RoboDK station: Sheet B.rdk

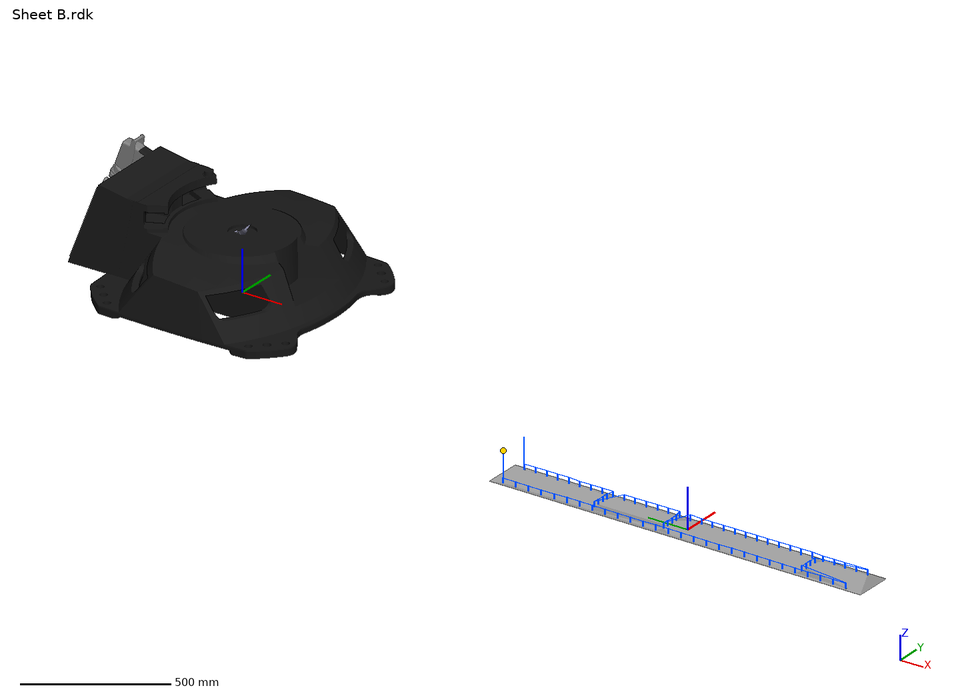
[picture v0: the station drawn from its stored meshes, robots at their saved joint values, targets as dots, program paths as lines]
Station Sheet B (saved by RoboDK 5.2.3). Poses are relative to the parent item; angles as X-Y-Z fixed-axis rotations.
  - frame KUKA KR 210 R2700 extra Base at (0, 0, 0) mm
    - robot KUKA KR 210 R2700 extra: 6 axes, payload 210 kg, reach 2696 mm, repeatability 0.06 mm, weight 1068 kg
        joint limits [-185, -140, -120, -350, -125, -350] to [185, -5, 155, 350, 125, 350]; home [0, -90, 90, 0, 0, 0]; saved at [-4.299, -27.561, 142.534, -183.011, 63.926, -182.019]
      - tool Spindle, TCP at (32, 0, 260) mm, rotated rx 0 ry 39 rz 0 deg, size 157.3 x 72 x 259.9 mm
  - frame Frame 2 at (1800, 0, -372.68) mm, rotated rx 0 ry 0 rz 90 deg
    - object Box 1 - Sheet B at (0, 0, 0) mm, size 148.8 x 1500 x 0.8 mm, geometry from Box 1 - Sheet B.stl
    - object Sheet B-box 1 Hole positioning at (0, 0, 0) mm, 72 curves, geometry from Point 72
  - machining project Point settings: rotZ(0) | rotX(0)*rotY(0) | rotz(0) | onStart | onPathStart | onApproach | onPoint | onRetract | onFinish | SetRPM(%1) | SetTool(%1) | Extruder(%1) | default | default | OutOnMov(%1) | OutOffMov(%1) | onPathFinish | M_RunCode(%1)
  - program Point (371 instructions, listed below)
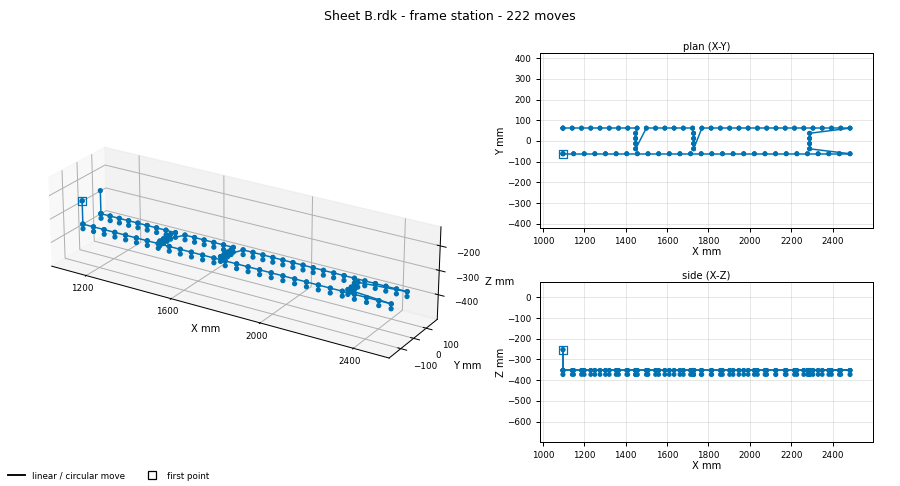
[picture p0: tool path of Sheet B.rdk in frame station, 222 of 222 moves have a stored position in this frame; points joined in program order, loops and branches not executed]

--- program Point (robot KUKA KR 210 R2700 extra) ---
  Smooth(1)
  Set speed (1000.0 mm/s)
  Set Ref.: Frame 2
  Set Tool: Spindle
  Show Spindle
  MoveJ 1 to (-61.9, 702.57, 120) mm, rotated rx 180 ry 0 rz 90 deg; joints [4.299, -27.561, 142.534, -176.989, 63.926, -177.981]
  MoveL 2 to (-61.9, 702.57, 120) mm, rotated rx 180 ry 0 rz 90 deg; joints [4.299, -27.561, 142.534, -176.989, 63.926, -177.981]
  MoveL 3 to (-61.9, 702.57, 20) mm, rotated rx -180 ry 0 rz 90 deg; joints [4.299, -20.368, 138.524, -177.064, 67.105, -177.799]
  MoveL 4 to (-61.9, 702.57, 20) mm, rotated rx -180 ry 0 rz 90 deg; joints [4.299, -20.368, 138.524, -177.064, 67.105, -177.799]
  Set speed (50.0 mm/s)
  MoveL 5 to (-61.9, 702.57, 0) mm, rotated rx 180 ry 0 rz 90 deg; joints [4.299, -19.028, 137.686, -177.075, 67.605, -177.771]
  MoveL 6 to (-61.9, 702.57, 20) mm, rotated rx -180 ry 0 rz 90 deg; joints [4.299, -20.368, 138.524, -177.064, 67.105, -177.799]
  Set speed (1000.0 mm/s)
  MoveL 7 to (-61.9, 651.24, 20) mm, rotated rx 180 ry 0 rz 90 deg; joints [4.048, -22.239, 136.879, -177.157, 63.598, -178.117]
  Set speed (50.0 mm/s)
  MoveL 8 to (-61.9, 651.24, 0) mm, rotated rx -180 ry 0 rz 90 deg; joints [4.048, -20.899, 136.068, -177.17, 64.126, -178.088]
  MoveL 9 to (-61.9, 651.24, 20) mm, rotated rx 180 ry 0 rz 90 deg; joints [4.048, -22.239, 136.879, -177.157, 63.598, -178.117]
  Set speed (1000.0 mm/s)
  MoveL 10 to (-61.9, 599.91, 20) mm, rotated rx 180 ry 0 rz 90 deg; joints [3.824, -23.844, 135.126, -177.229, 60.248, -178.402]
  Set speed (50.0 mm/s)
  MoveL 11 to (-61.9, 599.91, 0) mm, rotated rx -180 ry 0 rz 90 deg; joints [3.824, -22.512, 134.341, -177.244, 60.795, -178.372]
  MoveL 12 to (-61.9, 599.91, 20) mm, rotated rx 180 ry 0 rz 90 deg; joints [3.824, -23.844, 135.126, -177.229, 60.248, -178.402]
  Set speed (1000.0 mm/s)
  MoveL 13 to (-61.9, 548.57, 20) mm, rotated rx -180 ry 0 rz 90 deg; joints [3.624, -25.203, 133.273, -177.283, 57.044, -178.661]
  Set speed (50.0 mm/s)
  MoveL 14 to (-61.9, 548.57, 0) mm, rotated rx 180 ry 0 rz 90 deg; joints [3.624, -23.885, 132.514, -177.3, 57.602, -178.63]
  MoveL 15 to (-61.9, 548.57, 20) mm, rotated rx -180 ry 0 rz 90 deg; joints [3.624, -25.203, 133.273, -177.283, 57.044, -178.661]
  Set speed (1000.0 mm/s)
  MoveL 16 to (-61.9, 497.24, 20) mm, rotated rx 180 ry 0 rz 90 deg; joints [3.444, -26.333, 131.329, -177.321, 53.975, -178.899]
  Set speed (50.0 mm/s)
  MoveL 17 to (-61.9, 497.24, 0) mm, rotated rx -180 ry 0 rz 90 deg; joints [3.444, -25.033, 130.594, -177.34, 54.539, -178.866]
  MoveL 18 to (-61.9, 497.24, 20) mm, rotated rx 180 ry 0 rz 90 deg; joints [3.444, -26.333, 131.329, -177.321, 53.975, -178.899]
  Set speed (1000.0 mm/s)
  MoveL 19 to (-61.9, 445.91, 20) mm, rotated rx 180 ry 0 rz 90 deg; joints [3.28, -27.254, 129.3, -177.345, 51.03, -179.12]
  Set speed (50.0 mm/s)
  MoveL 20 to (-61.9, 445.91, 0) mm, rotated rx 180 ry 0 rz 90 deg; joints [3.28, -25.976, 128.588, -177.366, 51.595, -179.087]
  MoveL 21 to (-61.9, 445.91, 20) mm, rotated rx 180 ry 0 rz 90 deg; joints [3.28, -27.254, 129.3, -177.345, 51.03, -179.12]
  Set speed (1000.0 mm/s)
  MoveL 22 to (-61.9, 394.57, 20) mm, rotated rx -180 ry 0 rz 90 deg; joints [3.132, -27.982, 127.19, -177.357, 48.196, -179.328]
  Set speed (50.0 mm/s)
  MoveL 23 to (-61.9, 394.57, 0) mm, rotated rx 180 ry 0 rz 90 deg; joints [3.132, -26.729, 126.5, -177.379, 48.759, -179.294]
  MoveL 24 to (-61.9, 394.57, 20) mm, rotated rx -180 ry 0 rz 90 deg; joints [3.132, -27.982, 127.19, -177.357, 48.196, -179.328]
  Set speed (1000.0 mm/s)
  MoveL 25 to (-61.9, 343.24, 20) mm, rotated rx -180 ry 0 rz 90 deg; joints [2.996, -28.534, 125.006, -177.355, 45.464, -179.526]
  Set speed (50.0 mm/s)
  MoveL 26 to (-61.9, 343.24, 0) mm, rotated rx 180 ry 0 rz 90 deg; joints [2.996, -27.307, 124.335, -177.38, 46.02, -179.491]
  MoveL 27 to (-61.9, 343.24, 20) mm, rotated rx -180 ry 0 rz 90 deg; joints [2.996, -28.534, 125.006, -177.355, 45.464, -179.526]
  Set speed (1000.0 mm/s)
  MoveL 28 to (-61.9, 291.91, 20) mm, rotated rx -180 ry 0 rz 90 deg; joints [2.872, -28.924, 122.749, -177.341, 42.821, -179.718]
  Set speed (50.0 mm/s)
  MoveL 29 to (-61.9, 291.91, 0) mm, rotated rx 180 ry 0 rz 90 deg; joints [2.872, -27.723, 122.097, -177.369, 43.369, -179.681]
  MoveL 30 to (-61.9, 291.91, 20) mm, rotated rx -180 ry 0 rz 90 deg; joints [2.872, -28.924, 122.749, -177.341, 42.821, -179.718]
  Set speed (1000.0 mm/s)
  MoveL 31 to (-61.9, 240.57, 20) mm, rotated rx -180 ry 0 rz 90 deg; joints [2.757, -29.164, 120.423, -177.315, 40.257, -179.906]
  Set speed (50.0 mm/s)
  MoveL 32 to (-61.9, 240.57, 0) mm, rotated rx -180 ry 0 rz 90 deg; joints [2.757, -27.991, 119.788, -177.344, 40.795, -179.868]
  MoveL 33 to (-61.9, 240.57, 20) mm, rotated rx -180 ry 0 rz 90 deg; joints [2.757, -29.164, 120.423, -177.315, 40.257, -179.906]
  Set speed (1000.0 mm/s)
  MoveL 34 to (-61.9, 189.24, 20) mm, rotated rx 180 ry 0 rz 90 deg; joints [2.651, -29.267, 118.029, -177.275, 37.764, -180.093]
  Set speed (50.0 mm/s)
  MoveL 35 to (-61.9, 189.24, 0) mm, rotated rx -180 ry 0 rz 90 deg; joints [2.651, -28.12, 117.41, -177.307, 38.291, -180.053]
  MoveL 36 to (-61.9, 189.24, 20) mm, rotated rx 180 ry 0 rz 90 deg; joints [2.651, -29.267, 118.029, -177.275, 37.764, -180.093]
  Set speed (1000.0 mm/s)
  MoveL 37 to (-61.9, 137.91, 20) mm, rotated rx -180 ry 0 rz 90 deg; joints [2.553, -29.241, 115.568, -177.221, 35.331, -180.283]
  Set speed (50.0 mm/s)
  MoveL 38 to (-61.9, 137.91, 0) mm, rotated rx -180 ry 0 rz 90 deg; joints [2.553, -28.121, 114.963, -177.256, 35.846, -180.24]
  MoveL 39 to (-61.9, 137.91, 20) mm, rotated rx -180 ry 0 rz 90 deg; joints [2.553, -29.241, 115.568, -177.221, 35.331, -180.283]
  Set speed (1000.0 mm/s)
  MoveL 40 to (-61.9, 86.57, 20) mm, rotated rx 180 ry 0 rz 90 deg; joints [2.462, -29.097, 113.041, -177.151, 32.95, -180.478]
  Set speed (50.0 mm/s)
  MoveL 41 to (-61.9, 86.57, 0) mm, rotated rx -180 ry 0 rz 90 deg; joints [2.462, -28.002, 112.448, -177.188, 33.452, -180.432]
  MoveL 42 to (-61.9, 86.57, 20) mm, rotated rx 180 ry 0 rz 90 deg; joints [2.462, -29.097, 113.041, -177.151, 32.95, -180.478]
  Set speed (1000.0 mm/s)
  MoveL 43 to (-61.9, 35.24, 20) mm, rotated rx 180 ry 0 rz 90 deg; joints [2.378, -28.841, 110.446, -177.061, 30.614, -180.681]
  Set speed (50.0 mm/s)
  MoveL 44 to (-61.9, 35.24, 0) mm, rotated rx -180 ry 0 rz 90 deg; joints [2.378, -27.771, 109.865, -177.103, 31.102, -180.633]
  MoveL 45 to (-61.9, 35.24, 20) mm, rotated rx 180 ry 0 rz 90 deg; joints [2.378, -28.841, 110.446, -177.061, 30.614, -180.681]
  Set speed (1000.0 mm/s)
  MoveL 46 to (-61.9, -16.09, 20) mm, rotated rx 180 ry 0 rz 90 deg; joints [2.299, -28.479, 107.783, -176.949, 28.315, -180.899]
  Set speed (50.0 mm/s)
  MoveL 47 to (-61.9, -16.09, 0) mm, rotated rx -180 ry 0 rz 90 deg; joints [2.299, -27.434, 107.212, -176.996, 28.789, -180.847]
  MoveL 48 to (-61.9, -16.09, 20) mm, rotated rx 180 ry 0 rz 90 deg; joints [2.299, -28.479, 107.783, -176.949, 28.315, -180.899]
  Set speed (1000.0 mm/s)
  MoveL 49 to (-61.9, -67.43, 20) mm, rotated rx 180 ry 0 rz 90 deg; joints [2.225, -28.017, 105.049, -176.811, 26.045, -181.137]
  Set speed (50.0 mm/s)
  MoveL 50 to (-61.9, -67.43, 0) mm, rotated rx -180 ry 0 rz 90 deg; joints [2.225, -26.995, 104.487, -176.862, 26.505, -181.079]
  MoveL 51 to (-61.9, -67.43, 20) mm, rotated rx 180 ry 0 rz 90 deg; joints [2.225, -28.017, 105.049, -176.811, 26.045, -181.137]
  Set speed (1000.0 mm/s)
  MoveL 52 to (-61.9, -118.76, 20) mm, rotated rx -180 ry 0 rz 90 deg; joints [2.155, -27.459, 102.241, -176.637, 23.799, -181.402]
  Set speed (50.0 mm/s)
  MoveL 53 to (-61.9, -118.76, 0) mm, rotated rx -180 ry 0 rz 90 deg; joints [2.155, -26.459, 101.687, -176.696, 24.244, -181.338]
  MoveL 54 to (-61.9, -118.76, 20) mm, rotated rx -180 ry 0 rz 90 deg; joints [2.155, -27.459, 102.241, -176.637, 23.799, -181.402]
  Set speed (1000.0 mm/s)
  MoveL 55 to (-61.9, -170.09, 20) mm, rotated rx -180 ry 0 rz 90 deg; joints [2.09, -26.809, 99.357, -176.42, 21.568, -181.705]
  Set speed (50.0 mm/s)
  MoveL 56 to (-61.9, -170.09, 0) mm, rotated rx -180 ry 0 rz 90 deg; joints [2.09, -25.829, 98.809, -176.487, 21.998, -181.633]
  MoveL 57 to (-61.9, -170.09, 20) mm, rotated rx -180 ry 0 rz 90 deg; joints [2.09, -26.809, 99.357, -176.42, 21.568, -181.705]
  Set speed (1000.0 mm/s)
  MoveL 58 to (-61.9, -221.43, 20) mm, rotated rx 180 ry 0 rz 90 deg; joints [2.029, -26.067, 96.391, -176.144, 19.346, -182.062]
  Set speed (50.0 mm/s)
  MoveL 59 to (-61.9, -221.43, 0) mm, rotated rx 180 ry 0 rz 90 deg; joints [2.029, -25.107, 95.847, -176.222, 19.762, -181.979]
  MoveL 60 to (-61.9, -221.43, 20) mm, rotated rx 180 ry 0 rz 90 deg; joints [2.029, -26.067, 96.391, -176.144, 19.346, -182.062]
  Set speed (1000.0 mm/s)
  MoveL 61 to (-61.9, -272.76, 20) mm, rotated rx -180 ry 0 rz 90 deg; joints [1.971, -25.236, 93.337, -175.785, 17.128, -182.496]
  Set speed (50.0 mm/s)
  MoveL 62 to (-61.9, -272.76, 0) mm, rotated rx -180 ry 0 rz 90 deg; joints [1.971, -24.295, 92.797, -175.879, 17.528, -182.398]
  MoveL 63 to (-61.9, -272.76, 20) mm, rotated rx -180 ry 0 rz 90 deg; joints [1.971, -25.236, 93.337, -175.785, 17.128, -182.496]
  Set speed (1000.0 mm/s)
  MoveL 64 to (-61.9, -324.09, 20) mm, rotated rx -180 ry 0 rz 90 deg; joints [1.916, -24.316, 90.189, -175.307, 14.906, -183.046]
  Set speed (50.0 mm/s)
  MoveL 65 to (-61.9, -324.09, 0) mm, rotated rx -180 ry 0 rz 90 deg; joints [1.916, -23.391, 89.651, -175.423, 15.29, -182.926]
  MoveL 66 to (-61.9, -324.09, 20) mm, rotated rx -180 ry 0 rz 90 deg; joints [1.916, -24.316, 90.189, -175.307, 14.906, -183.046]
  Set speed (1000.0 mm/s)
  MoveL 67 to (-61.9, -375.43, 20) mm, rotated rx 180 ry 0 rz 90 deg; joints [1.865, -23.305, 86.938, -174.644, 12.672, -183.777]
  Set speed (50.0 mm/s)
  MoveL 68 to (-61.9, -375.43, 0) mm, rotated rx -180 ry 0 rz 90 deg; joints [1.865, -22.396, 86.4, -174.793, 13.041, -183.624]
  MoveL 69 to (-61.9, -375.43, 20) mm, rotated rx 180 ry 0 rz 90 deg; joints [1.865, -23.305, 86.938, -174.644, 12.672, -183.777]
  Set speed (1000.0 mm/s)
  MoveL 70 to (-61.9, -426.76, 20) mm, rotated rx -180 ry 0 rz 90 deg; joints [1.816, -22.202, 83.574, -173.671, 10.421, -184.814]
  Set speed (50.0 mm/s)
  MoveL 71 to (-61.9, -426.76, 0) mm, rotated rx 180 ry 0 rz 90 deg; joints [1.816, -21.307, 83.035, -173.877, 10.774, -184.605]
  MoveL 72 to (-61.9, -426.76, 20) mm, rotated rx -180 ry 0 rz 90 deg; joints [1.816, -22.202, 83.574, -173.671, 10.421, -184.814]
  Set speed (1000.0 mm/s)
  MoveL 73 to (-61.9, -478.09, 20) mm, rotated rx 180 ry 0 rz 90 deg; joints [1.769, -21.002, 80.085, -172.118, 8.145, -186.428]
  Set speed (50.0 mm/s)
  MoveL 74 to (-61.9, -478.09, 0) mm, rotated rx -180 ry 0 rz 90 deg; joints [1.769, -20.12, 79.541, -172.43, 8.481, -186.113]
  MoveL 75 to (-61.9, -478.09, 20) mm, rotated rx 180 ry 0 rz 90 deg; joints [1.769, -21.002, 80.085, -172.118, 8.145, -186.428]
  Set speed (1000.0 mm/s)
  MoveL 76 to (-61.9, -529.43, 20) mm, rotated rx -180 ry 0 rz 90 deg; joints [1.725, -19.7, 76.453, -169.273, 5.842, -189.332]
  Set speed (50.0 mm/s)
  MoveL 77 to (-61.9, -529.43, 0) mm, rotated rx 180 ry 0 rz 90 deg; joints [1.725, -18.828, 75.903, -169.828, 6.158, -188.774]
  MoveL 78 to (-61.9, -529.43, 20) mm, rotated rx -180 ry 0 rz 90 deg; joints [1.725, -19.7, 76.453, -169.273, 5.842, -189.332]
  Set speed (1000.0 mm/s)
  MoveL 79 to (-61.9, -580.76, 20) mm, rotated rx -180 ry 0 rz 90 deg; joints [1.683, -18.288, 72.66, -162.494, 3.523, -196.167]
  Set speed (50.0 mm/s)
  MoveL 80 to (-61.9, -580.76, 0) mm, rotated rx 180 ry 0 rz 90 deg; joints [1.683, -17.425, 72.101, -163.866, 3.814, -194.792]
  MoveL 81 to (-61.9, -580.76, 20) mm, rotated rx -180 ry 0 rz 90 deg; joints [1.683, -18.288, 72.66, -162.494, 3.523, -196.167]
  Set speed (1000.0 mm/s)
  MoveL 82 to (-61.9, -632.09, 20) mm, rotated rx -180 ry 0 rz 70 deg; joints [-0.839, -16.255, 67.408, -277.48, 13.05, -98.802]
  Set speed (50.0 mm/s)
  MoveL 83 to (-61.9, -632.09, 0) mm, rotated rx -180 ry 0 rz 70 deg; joints [-0.839, -15.4, 66.832, -276.285, 13.016, -100.029]
  MoveL 84 to (-61.9, -632.09, 20) mm, rotated rx -180 ry 0 rz 70 deg; joints [-0.839, -16.255, 67.408, -277.48, 13.05, -98.802]
  Set speed (1000.0 mm/s)
  MoveL 85 to (-61.9, -683.43, 20) mm, rotated rx -180 ry 0 rz 70 deg; joints [-0.819, -14.541, 63.132, -288.04, 13.606, -87.937]
  Set speed (50.0 mm/s)
  MoveL 86 to (-61.9, -683.43, 0) mm, rotated rx -180 ry 0 rz 70 deg; joints [-0.819, -13.689, 62.537, -287.023, 13.528, -88.983]
  MoveL 87 to (-61.9, -683.43, 20) mm, rotated rx -180 ry 0 rz 70 deg; joints [-0.819, -14.541, 63.132, -288.04, 13.606, -87.937]
  Set speed (1000.0 mm/s)
  MoveL 88 to (-38, -488.43, 20) mm, rotated rx 180 ry 0 rz 90 deg; joints [1.081, -20.763, 79.407, -174.897, 7.669, -184.218]
  Set speed (50.0 mm/s)
  MoveL 89 to (-38, -488.43, 0) mm, rotated rx 180 ry 0 rz 90 deg; joints [1.081, -19.883, 78.862, -175.109, 8.003, -184.003]
  MoveL 90 to (-38, -488.43, 20) mm, rotated rx -180 ry 0 rz 90 deg; joints [1.081, -20.763, 79.407, -174.897, 7.669, -184.218]
  Set speed (1000.0 mm/s)
  MoveL 91 to (-13, -488.43, 20) mm, rotated rx 180 ry 0 rz 90 deg; joints [0.37, -20.771, 79.429, -178.254, 7.661, -181.443]
  Set speed (50.0 mm/s)
  MoveL 92 to (-13, -488.43, 0) mm, rotated rx -180 ry 0 rz 90 deg; joints [0.37, -19.89, 78.884, -178.327, 7.997, -181.369]
  MoveL 93 to (-13, -488.43, 20) mm, rotated rx 180 ry 0 rz 90 deg; joints [0.37, -20.771, 79.429, -178.254, 7.661, -181.443]
  Set speed (1000.0 mm/s)
  MoveL 94 to (12, -488.43, 20) mm, rotated rx -180 ry 0 rz 90 deg; joints [-0.341, -20.771, 79.429, -181.611, 7.661, -178.668]
  Set speed (50.0 mm/s)
  MoveL 95 to (12, -488.43, 0) mm, rotated rx -180 ry 0 rz 90 deg; joints [-0.341, -19.891, 78.885, -181.544, 7.996, -178.736]
  MoveL 96 to (12, -488.43, 20) mm, rotated rx -180 ry 0 rz 90 deg; joints [-0.341, -20.771, 79.429, -181.611, 7.661, -178.668]
  Set speed (1000.0 mm/s)
  MoveL 97 to (37, -488.43, 20) mm, rotated rx -180 ry 0 rz 90 deg; joints [-1.052, -20.763, 79.408, -184.969, 7.668, -175.893]
  Set speed (50.0 mm/s)
  MoveL 98 to (37, -488.43, 0) mm, rotated rx -180 ry 0 rz 90 deg; joints [-1.052, -19.883, 78.863, -184.762, 8.003, -176.102]
  MoveL 99 to (37, -488.43, 20) mm, rotated rx -180 ry 0 rz 90 deg; joints [-1.052, -20.763, 79.408, -184.969, 7.668, -175.893]
  Set speed (1000.0 mm/s)
  MoveL 100 to (61.9, -683.43, 20) mm, rotated rx -180 ry 0 rz 70 deg; joints [-4, -14.358, 62.684, -288.833, 15.691, -89.578]
  Set speed (50.0 mm/s)
  MoveL 101 to (61.9, -683.43, 0) mm, rotated rx -180 ry 0 rz 70 deg; joints [-4, -13.506, 62.087, -287.969, 15.61, -90.475]
  MoveL 102 to (61.9, -683.43, 20) mm, rotated rx 180 ry 0 rz 70 deg; joints [-4, -14.358, 62.684, -288.833, 15.691, -89.578]
  Set speed (1000.0 mm/s)
  MoveL 103 to (61.9, -638.72, 20) mm, rotated rx -180 ry 0 rz 70 deg; joints [-4.081, -15.87, 66.435, -280.993, 15.164, -97.774]
  Set speed (50.0 mm/s)
  MoveL 104 to (61.9, -638.72, 0) mm, rotated rx -180 ry 0 rz 70 deg; joints [-4.081, -15.016, 65.855, -279.998, 15.114, -98.805]
  MoveL 105 to (61.9, -638.72, 20) mm, rotated rx -180 ry 0 rz 70 deg; joints [-4.081, -15.87, 66.435, -280.993, 15.164, -97.774]
  Set speed (1000.0 mm/s)
  MoveL 106 to (61.9, -594.01, 20) mm, rotated rx 180 ry 0 rz 90 deg; joints [-1.672, -17.905, 71.652, -201.052, 2.931, -160.273]
  Set speed (50.0 mm/s)
  MoveL 107 to (61.9, -594.01, 0) mm, rotated rx -180 ry 0 rz 90 deg; joints [-1.672, -17.044, 71.09, -199.137, 3.212, -162.191]
  MoveL 108 to (61.9, -594.01, 20) mm, rotated rx -180 ry 0 rz 90 deg; joints [-1.672, -17.905, 71.652, -201.052, 2.931, -160.273]
  Set speed (1000.0 mm/s)
  MoveL 109 to (61.9, -549.3, 20) mm, rotated rx 180 ry 0 rz 90 deg; joints [-1.709, -19.167, 75.005, -192.575, 4.944, -168.798]
  Set speed (50.0 mm/s)
  MoveL 110 to (61.9, -549.3, 0) mm, rotated rx 180 ry 0 rz 90 deg; joints [-1.709, -18.299, 74.452, -191.829, 5.252, -169.547]
  MoveL 111 to (61.9, -549.3, 20) mm, rotated rx 180 ry 0 rz 90 deg; joints [-1.709, -19.167, 75.005, -192.575, 4.944, -168.798]
  Set speed (1000.0 mm/s)
  MoveL 112 to (61.9, -504.59, 20) mm, rotated rx -180 ry 0 rz 90 deg; joints [-1.746, -20.343, 78.229, -189.105, 6.96, -172.318]
  Set speed (50.0 mm/s)
  MoveL 113 to (61.9, -504.59, 0) mm, rotated rx 180 ry 0 rz 90 deg; joints [-1.746, -19.466, 77.682, -188.697, 7.286, -172.729]
  MoveL 114 to (61.9, -504.59, 20) mm, rotated rx -180 ry 0 rz 90 deg; joints [-1.746, -20.343, 78.229, -189.105, 6.96, -172.318]
  Set speed (1000.0 mm/s)
  MoveL 115 to (61.9, -459.88, 20) mm, rotated rx -180 ry 0 rz 90 deg; joints [-1.785, -21.439, 81.338, -187.236, 8.956, -174.239]
  Set speed (50.0 mm/s)
  MoveL 116 to (61.9, -459.88, 0) mm, rotated rx 180 ry 0 rz 90 deg; joints [-1.785, -20.552, 80.796, -186.971, 9.298, -174.508]
  MoveL 117 to (61.9, -459.88, 20) mm, rotated rx -180 ry 0 rz 90 deg; joints [-1.785, -21.439, 81.338, -187.236, 8.956, -174.239]
  Set speed (1000.0 mm/s)
  MoveL 118 to (61.9, -415.17, 20) mm, rotated rx 180 ry 0 rz 90 deg; joints [-1.826, -22.459, 84.344, -186.072, 10.931, -175.457]
  Set speed (50.0 mm/s)
  MoveL 119 to (61.9, -415.17, 0) mm, rotated rx -180 ry 0 rz 90 deg; joints [-1.826, -21.561, 83.805, -185.882, 11.288, -175.651]
  MoveL 120 to (61.9, -415.17, 20) mm, rotated rx 180 ry 0 rz 90 deg; joints [-1.826, -22.459, 84.344, -186.072, 10.931, -175.457]
  Set speed (1000.0 mm/s)
  MoveL 121 to (61.9, -370.46, 20) mm, rotated rx 180 ry 0 rz 90 deg; joints [-1.87, -23.407, 87.258, -185.281, 12.889, -176.304]
  Set speed (50.0 mm/s)
  MoveL 122 to (61.9, -370.46, 0) mm, rotated rx -180 ry 0 rz 90 deg; joints [-1.87, -22.497, 86.72, -185.136, 13.259, -176.454]
  MoveL 123 to (61.9, -370.46, 20) mm, rotated rx 180 ry 0 rz 90 deg; joints [-1.87, -23.407, 87.258, -185.281, 12.889, -176.304]
  Set speed (1000.0 mm/s)
  MoveL 124 to (61.9, -325.75, 20) mm, rotated rx -180 ry 0 rz 90 deg; joints [-1.915, -24.285, 90.086, -184.711, 14.834, -176.934]
  Set speed (50.0 mm/s)
  MoveL 125 to (61.9, -325.75, 0) mm, rotated rx 180 ry 0 rz 90 deg; joints [-1.915, -23.361, 89.548, -184.594, 15.218, -177.054]
  MoveL 126 to (61.9, -325.75, 20) mm, rotated rx -180 ry 0 rz 90 deg; joints [-1.915, -24.285, 90.086, -184.711, 14.834, -176.934]
  Set speed (1000.0 mm/s)
  MoveL 127 to (61.9, -281.04, 20) mm, rotated rx -180 ry 0 rz 90 deg; joints [-1.962, -25.094, 92.836, -184.282, 16.77, -177.424]
  Set speed (50.0 mm/s)
  MoveL 128 to (61.9, -281.04, 0) mm, rotated rx 180 ry 0 rz 90 deg; joints [-1.962, -24.155, 92.296, -184.186, 17.168, -177.525]
  MoveL 129 to (61.9, -281.04, 20) mm, rotated rx -180 ry 0 rz 90 deg; joints [-1.962, -25.094, 92.836, -184.282, 16.77, -177.424]
  Set speed (1000.0 mm/s)
  MoveL 130 to (61.9, -236.33, 20) mm, rotated rx -180 ry 0 rz 90 deg; joints [-2.012, -25.835, 95.514, -183.95, 18.703, -177.821]
  Set speed (50.0 mm/s)
  MoveL 131 to (61.9, -236.33, 0) mm, rotated rx 180 ry 0 rz 90 deg; joints [-2.012, -24.881, 94.971, -183.868, 19.114, -177.908]
  MoveL 132 to (61.9, -236.33, 20) mm, rotated rx -180 ry 0 rz 90 deg; joints [-2.012, -25.835, 95.514, -183.95, 18.703, -177.821]
  Set speed (1000.0 mm/s)
  MoveL 133 to (61.9, -191.62, 20) mm, rotated rx -180 ry 0 rz 90 deg; joints [-2.064, -26.509, 98.123, -183.687, 20.636, -178.153]
  Set speed (50.0 mm/s)
  MoveL 134 to (61.9, -191.62, 0) mm, rotated rx -180 ry 0 rz 90 deg; joints [-2.064, -25.538, 97.577, -183.616, 21.06, -178.229]
  MoveL 135 to (61.9, -191.62, 20) mm, rotated rx -180 ry 0 rz 90 deg; joints [-2.064, -26.509, 98.123, -183.687, 20.636, -178.153]
  Set speed (1000.0 mm/s)
  MoveL 136 to (61.9, -146.91, 20) mm, rotated rx 180 ry 0 rz 90 deg; joints [-2.119, -27.114, 100.669, -183.475, 22.574, -178.437]
  Set speed (50.0 mm/s)
  MoveL 137 to (61.9, -146.91, 0) mm, rotated rx -180 ry 0 rz 90 deg; joints [-2.119, -26.125, 100.119, -183.413, 23.011, -178.505]
  MoveL 138 to (61.9, -146.91, 20) mm, rotated rx 180 ry 0 rz 90 deg; joints [-2.119, -27.114, 100.669, -183.475, 22.574, -178.437]
  Set speed (1000.0 mm/s)
  MoveL 139 to (61.9, -102.2, 20) mm, rotated rx -180 ry 0 rz 90 deg; joints [-2.177, -27.649, 103.155, -183.302, 24.521, -178.687]
  Set speed (50.0 mm/s)
  MoveL 140 to (61.9, -102.2, 0) mm, rotated rx -180 ry 0 rz 90 deg; joints [-2.177, -26.642, 102.599, -183.247, 24.971, -178.749]
  MoveL 141 to (61.9, -102.2, 20) mm, rotated rx -180 ry 0 rz 90 deg; joints [-2.177, -27.649, 103.155, -183.302, 24.521, -178.687]
  Set speed (1000.0 mm/s)
  MoveL 142 to (61.9, -57.49, 20) mm, rotated rx -180 ry 0 rz 90 deg; joints [-2.239, -28.114, 105.584, -183.16, 26.483, -178.911]
  Set speed (50.0 mm/s)
  MoveL 143 to (61.9, -57.49, 0) mm, rotated rx -180 ry 0 rz 90 deg; joints [-2.239, -27.088, 105.02, -183.11, 26.945, -178.967]
  MoveL 144 to (61.9, -57.49, 20) mm, rotated rx -180 ry 0 rz 90 deg; joints [-2.239, -28.114, 105.584, -183.16, 26.483, -178.911]
  Set speed (1000.0 mm/s)
  MoveL 145 to (61.9, -12.78, 20) mm, rotated rx -180 ry 0 rz 90 deg; joints [-2.304, -28.505, 107.957, -183.043, 28.463, -179.115]
  Set speed (50.0 mm/s)
  MoveL 146 to (61.9, -12.78, 0) mm, rotated rx 180 ry 0 rz 90 deg; joints [-2.304, -27.459, 107.385, -182.997, 28.937, -179.167]
  MoveL 147 to (61.9, -12.78, 20) mm, rotated rx -180 ry 0 rz 90 deg; joints [-2.304, -28.505, 107.957, -183.043, 28.463, -179.115]
  Set speed (1000.0 mm/s)
  MoveL 148 to (61.9, 31.93, 20) mm, rotated rx 180 ry 0 rz 90 deg; joints [-2.373, -28.82, 110.276, -182.945, 30.465, -179.305]
  Set speed (50.0 mm/s)
  MoveL 149 to (61.9, 31.93, 0) mm, rotated rx -180 ry 0 rz 90 deg; joints [-2.373, -27.753, 109.696, -182.903, 30.952, -179.354]
  MoveL 150 to (61.9, 31.93, 20) mm, rotated rx 180 ry 0 rz 90 deg; joints [-2.373, -28.82, 110.276, -182.945, 30.465, -179.305]
  Set speed (1000.0 mm/s)
  MoveL 151 to (-38, 71.57, 20) mm, rotated rx -180 ry 0 rz 90 deg; joints [1.497, -29.037, 112.331, -178.237, 32.296, -180.327]
  Set speed (50.0 mm/s)
  MoveL 152 to (-38, 71.57, 0) mm, rotated rx 180 ry 0 rz 90 deg; joints [1.497, -27.95, 111.742, -178.261, 32.795, -180.299]
  MoveL 153 to (-38, 71.57, 20) mm, rotated rx -180 ry 0 rz 90 deg; joints [1.497, -29.037, 112.331, -178.237, 32.296, -180.327]
  Set speed (1000.0 mm/s)
  MoveL 154 to (-13, 71.57, 20) mm, rotated rx 180 ry 0 rz 90 deg; joints [0.512, -29.039, 112.353, -179.397, 32.314, -180.112]
  Set speed (50.0 mm/s)
  MoveL 155 to (-13, 71.57, 0) mm, rotated rx -180 ry 0 rz 90 deg; joints [0.512, -27.951, 111.764, -179.405, 32.813, -180.102]
  MoveL 156 to (-13, 71.57, 20) mm, rotated rx 180 ry 0 rz 90 deg; joints [0.512, -29.039, 112.353, -179.397, 32.314, -180.112]
  Set speed (1000.0 mm/s)
  MoveL 157 to (12, 71.57, 20) mm, rotated rx 180 ry 0 rz 90 deg; joints [-0.473, -29.039, 112.353, -180.557, 32.315, -179.897]
  Set speed (50.0 mm/s)
  MoveL 158 to (12, 71.57, 0) mm, rotated rx 180 ry 0 rz 90 deg; joints [-0.473, -27.951, 111.764, -180.549, 32.813, -179.906]
  MoveL 159 to (12, 71.57, 20) mm, rotated rx 180 ry 0 rz 90 deg; joints [-0.473, -29.039, 112.353, -180.557, 32.315, -179.897]
  Set speed (1000.0 mm/s)
  MoveL 160 to (37, 71.57, 20) mm, rotated rx -180 ry 0 rz 90 deg; joints [-1.457, -29.037, 112.332, -181.717, 32.298, -179.682]
  Set speed (50.0 mm/s)
  MoveL 161 to (37, 71.57, 0) mm, rotated rx -180 ry 0 rz 90 deg; joints [-1.457, -27.95, 111.743, -181.693, 32.796, -179.709]
  MoveL 162 to (37, 71.57, 20) mm, rotated rx -180 ry 0 rz 90 deg; joints [-1.457, -29.037, 112.332, -181.717, 32.298, -179.682]
  Set speed (1000.0 mm/s)
  MoveL 163 to (61.9, 76.64, 20) mm, rotated rx 180 ry 0 rz 90 deg; joints [-2.446, -29.056, 112.544, -182.865, 32.495, -179.484]
  Set speed (50.0 mm/s)
  MoveL 164 to (61.9, 76.64, 0) mm, rotated rx -180 ry 0 rz 90 deg; joints [-2.446, -27.966, 111.954, -182.827, 32.994, -179.53]
  MoveL 165 to (61.9, 76.64, 20) mm, rotated rx 180 ry 0 rz 90 deg; joints [-2.446, -29.056, 112.544, -182.865, 32.495, -179.484]
  Set speed (1000.0 mm/s)
  MoveL 166 to (61.9, 121.35, 20) mm, rotated rx -180 ry 0 rz 90 deg; joints [-2.523, -29.207, 114.76, -182.8, 34.558, -179.655]
  Set speed (50.0 mm/s)
  MoveL 167 to (61.9, 121.35, 0) mm, rotated rx -180 ry 0 rz 90 deg; joints [-2.523, -28.096, 114.16, -182.764, 35.068, -179.699]
  MoveL 168 to (61.9, 121.35, 20) mm, rotated rx -180 ry 0 rz 90 deg; joints [-2.523, -29.207, 114.76, -182.8, 34.558, -179.655]
  Set speed (1000.0 mm/s)
  MoveL 169 to (61.9, 166.06, 20) mm, rotated rx 180 ry 0 rz 90 deg; joints [-2.606, -29.271, 116.926, -182.747, 36.658, -179.822]
  Set speed (50.0 mm/s)
  MoveL 170 to (61.9, 166.06, 0) mm, rotated rx -180 ry 0 rz 90 deg; joints [-2.606, -28.136, 116.313, -182.714, 37.18, -179.863]
  MoveL 171 to (61.9, 166.06, 20) mm, rotated rx 180 ry 0 rz 90 deg; joints [-2.606, -29.271, 116.926, -182.747, 36.658, -179.822]
  Set speed (1000.0 mm/s)
  MoveL 172 to (61.9, 210.77, 20) mm, rotated rx -180 ry 0 rz 90 deg; joints [-2.695, -29.24, 119.041, -182.706, 38.802, -179.985]
  Set speed (50.0 mm/s)
  MoveL 173 to (61.9, 210.77, 0) mm, rotated rx -180 ry 0 rz 90 deg; joints [-2.695, -28.082, 118.416, -182.676, 39.333, -180.025]
  MoveL 174 to (61.9, 210.77, 20) mm, rotated rx -180 ry 0 rz 90 deg; joints [-2.695, -29.24, 119.041, -182.706, 38.802, -179.985]
  Set speed (1000.0 mm/s)
  MoveL 175 to (61.9, 255.48, 20) mm, rotated rx -180 ry 0 rz 90 deg; joints [-2.789, -29.109, 121.106, -182.676, 40.994, -180.148]
  Set speed (50.0 mm/s)
  MoveL 176 to (61.9, 255.48, 0) mm, rotated rx -180 ry 0 rz 90 deg; joints [-2.789, -27.928, 120.466, -182.647, 41.535, -180.186]
  MoveL 177 to (61.9, 255.48, 20) mm, rotated rx -180 ry 0 rz 90 deg; joints [-2.789, -29.109, 121.106, -182.676, 40.994, -180.148]
  Set speed (1000.0 mm/s)
  MoveL 178 to (61.9, 300.19, 20) mm, rotated rx -180 ry 0 rz 90 deg; joints [-2.891, -28.871, 123.118, -182.655, 43.242, -180.312]
  Set speed (50.0 mm/s)
  MoveL 179 to (61.9, 300.19, 0) mm, rotated rx -180 ry 0 rz 90 deg; joints [-2.891, -27.666, 122.463, -182.629, 43.791, -180.349]
  MoveL 180 to (61.9, 300.19, 20) mm, rotated rx -180 ry 0 rz 90 deg; joints [-2.891, -28.871, 123.118, -182.655, 43.242, -180.312]
  Set speed (1000.0 mm/s)
  MoveL 181 to (-38, 351.57, 20) mm, rotated rx 180 ry 0 rz 90 deg; joints [1.853, -28.446, 125.409, -178.378, 45.96, -179.688]
  Set speed (50.0 mm/s)
  MoveL 182 to (-38, 351.57, 0) mm, rotated rx -180 ry 0 rz 90 deg; joints [1.853, -27.214, 124.735, -178.393, 46.518, -179.666]
  MoveL 183 to (-38, 351.57, 20) mm, rotated rx 180 ry 0 rz 90 deg; joints [1.853, -28.446, 125.409, -178.378, 45.96, -179.688]
  Set speed (1000.0 mm/s)
  MoveL 184 to (-13, 351.57, 20) mm, rotated rx 180 ry 0 rz 90 deg; joints [0.634, -28.441, 125.432, -179.445, 45.991, -179.893]
  Set speed (50.0 mm/s)
  MoveL 185 to (-13, 351.57, 0) mm, rotated rx 180 ry 0 rz 90 deg; joints [0.634, -27.208, 124.758, -179.45, 46.549, -179.885]
  MoveL 186 to (-13, 351.57, 20) mm, rotated rx 180 ry 0 rz 90 deg; joints [0.634, -28.441, 125.432, -179.445, 45.991, -179.893]
  Set speed (1000.0 mm/s)
  MoveL 187 to (12, 351.57, 20) mm, rotated rx -180 ry 0 rz 90 deg; joints [-0.585, -28.441, 125.433, -180.512, 45.992, -180.099]
  Set speed (50.0 mm/s)
  MoveL 188 to (12, 351.57, 0) mm, rotated rx 180 ry 0 rz 90 deg; joints [-0.585, -27.208, 124.759, -180.507, 46.55, -180.106]
  MoveL 189 to (12, 351.57, 20) mm, rotated rx -180 ry 0 rz 90 deg; joints [-0.585, -28.441, 125.433, -180.512, 45.992, -180.099]
  Set speed (1000.0 mm/s)
  MoveL 190 to (37, 351.57, 20) mm, rotated rx 180 ry 0 rz 90 deg; joints [-1.805, -28.446, 125.41, -181.58, 45.962, -180.304]
  Set speed (50.0 mm/s)
  MoveL 191 to (37, 351.57, 0) mm, rotated rx -180 ry 0 rz 90 deg; joints [-1.805, -27.214, 124.736, -181.565, 46.519, -180.326]
  MoveL 192 to (37, 351.57, 20) mm, rotated rx 180 ry 0 rz 90 deg; joints [-1.805, -28.446, 125.41, -181.58, 45.962, -180.304]
  Set speed (1000.0 mm/s)
  MoveL 193 to (61.9, 344.89, 20) mm, rotated rx 180 ry 0 rz 90 deg; joints [-3, -28.519, 125.077, -182.645, 45.55, -180.48]
  Set speed (50.0 mm/s)
  MoveL 194 to (61.9, 344.89, 0) mm, rotated rx 180 ry 0 rz 90 deg; joints [-3, -27.291, 124.406, -182.62, 46.107, -180.515]
  MoveL 195 to (61.9, 344.89, 20) mm, rotated rx 180 ry 0 rz 90 deg; joints [-3, -28.519, 125.077, -182.645, 45.55, -180.48]
  Set speed (1000.0 mm/s)
  MoveL 196 to (61.9, 389.6, 20) mm, rotated rx 180 ry 0 rz 90 deg; joints [-3.118, -28.043, 126.982, -182.643, 47.928, -180.652]
  Set speed (50.0 mm/s)
  MoveL 197 to (61.9, 389.6, 0) mm, rotated rx -180 ry 0 rz 90 deg; joints [-3.118, -26.792, 126.293, -182.62, 48.489, -180.687]
  MoveL 198 to (61.9, 389.6, 20) mm, rotated rx 180 ry 0 rz 90 deg; joints [-3.118, -28.043, 126.982, -182.643, 47.928, -180.652]
  Set speed (1000.0 mm/s)
  MoveL 199 to (61.9, 434.31, 20) mm, rotated rx -180 ry 0 rz 90 deg; joints [-3.245, -27.435, 128.83, -182.651, 50.38, -180.832]
  Set speed (50.0 mm/s)
  MoveL 200 to (61.9, 434.31, 0) mm, rotated rx -180 ry 0 rz 90 deg; joints [-3.245, -26.162, 128.123, -182.63, 50.945, -180.866]
  MoveL 201 to (61.9, 434.31, 20) mm, rotated rx -180 ry 0 rz 90 deg; joints [-3.245, -27.435, 128.83, -182.651, 50.38, -180.832]
  Set speed (1000.0 mm/s)
  MoveL 202 to (61.9, 479.02, 20) mm, rotated rx 180 ry 0 rz 90 deg; joints [-3.384, -26.683, 130.618, -182.669, 52.916, -181.021]
  Set speed (50.0 mm/s)
  MoveL 203 to (61.9, 479.02, 0) mm, rotated rx -180 ry 0 rz 90 deg; joints [-3.384, -25.391, 129.892, -182.649, 53.481, -181.054]
  MoveL 204 to (61.9, 479.02, 20) mm, rotated rx 180 ry 0 rz 90 deg; joints [-3.384, -26.683, 130.618, -182.669, 52.916, -181.021]
  Set speed (1000.0 mm/s)
  MoveL 205 to (61.9, 523.73, 20) mm, rotated rx 180 ry 0 rz 90 deg; joints [-3.534, -25.777, 132.343, -182.697, 55.543, -181.221]
  Set speed (50.0 mm/s)
  MoveL 206 to (61.9, 523.73, 0) mm, rotated rx 180 ry 0 rz 90 deg; joints [-3.534, -24.467, 131.596, -182.679, 56.104, -181.253]
  MoveL 207 to (61.9, 523.73, 20) mm, rotated rx 180 ry 0 rz 90 deg; joints [-3.534, -25.777, 132.343, -182.697, 55.543, -181.221]
  Set speed (1000.0 mm/s)
  MoveL 208 to (61.9, 568.44, 20) mm, rotated rx -180 ry 0 rz 90 deg; joints [-3.699, -24.705, 134.001, -182.736, 58.267, -181.436]
  Set speed (50.0 mm/s)
  MoveL 209 to (61.9, 568.44, 0) mm, rotated rx -180 ry 0 rz 90 deg; joints [-3.699, -23.381, 133.233, -182.72, 58.822, -181.467]
  MoveL 210 to (61.9, 568.44, 20) mm, rotated rx -180 ry 0 rz 90 deg; joints [-3.699, -24.705, 134.001, -182.736, 58.267, -181.436]
  Set speed (1000.0 mm/s)
  MoveL 211 to (61.9, 613.15, 20) mm, rotated rx -180 ry 0 rz 90 deg; joints [-3.88, -23.455, 135.588, -182.788, 61.098, -181.669]
  Set speed (50.0 mm/s)
  MoveL 212 to (61.9, 613.15, 0) mm, rotated rx 180 ry 0 rz 90 deg; joints [-3.88, -22.12, 134.797, -182.773, 61.641, -181.699]
  MoveL 213 to (61.9, 613.15, 20) mm, rotated rx -180 ry 0 rz 90 deg; joints [-3.88, -23.455, 135.588, -182.788, 61.098, -181.669]
  Set speed (1000.0 mm/s)
  MoveL 214 to (61.9, 657.86, 20) mm, rotated rx 180 ry 0 rz 90 deg; joints [-4.079, -22.013, 137.097, -182.854, 64.041, -181.922]
  Set speed (50.0 mm/s)
  MoveL 215 to (61.9, 657.86, 0) mm, rotated rx -180 ry 0 rz 90 deg; joints [-4.079, -20.673, 136.283, -182.841, 64.567, -181.951]
  MoveL 216 to (61.9, 657.86, 20) mm, rotated rx 180 ry 0 rz 90 deg; joints [-4.079, -22.013, 137.097, -182.854, 64.041, -181.922]
  Set speed (1000.0 mm/s)
  MoveL 217 to (61.9, 702.57, 20) mm, rotated rx 180 ry 0 rz 90 deg; joints [-4.299, -20.368, 138.524, -182.936, 67.105, -182.201]
  Set speed (50.0 mm/s)
  MoveL 218 to (61.9, 702.57, 0) mm, rotated rx -180 ry 0 rz 90 deg; joints [-4.299, -19.028, 137.686, -182.925, 67.605, -182.229]
  MoveL 219 to (61.9, 702.57, 20) mm, rotated rx 180 ry 0 rz 90 deg; joints [-4.299, -20.368, 138.524, -182.936, 67.105, -182.201]
  MoveL 220 to (61.9, 702.57, 20) mm, rotated rx 180 ry 0 rz 90 deg; joints [-4.299, -20.368, 138.524, -182.936, 67.105, -182.201]
  Set speed (1000.0 mm/s)
  MoveL 221 to (61.9, 702.57, 20) mm, rotated rx 180 ry 0 rz 90 deg; joints [-4.299, -20.368, 138.524, -182.936, 67.105, -182.201]
  MoveL 222 to (61.9, 702.57, 120) mm, rotated rx -180 ry 0 rz 90 deg; joints [-4.299, -27.561, 142.534, -183.011, 63.926, -182.019]
